// TwinCAT 3 PLC project Publisher
// ProgramVersion: 3.1.4022.0
// libraries:
//   Tc2_Standard, * (Beckhoff Automation GmbH)
//   Tc2_System, * (Beckhoff Automation GmbH)
//   Tc3_EventLogger, * (Beckhoff Automation GmbH)
//   Tc3_Module, * (Beckhoff Automation GmbH)
// project tree:
//   / PublisherTask.TcTTO (not stored)
//   POUs/ MAIN.TcPOU
// real-time tasks:
//   TASK PublisherTask: cycle T#10ms, priority 20, ADS port 350
//   TASK ListenerTask: cycle T#10ms, priority 1, ADS port 351

// ---- POUs/MAIN.TcPOU
PROGRAM MAIN
VAR
	bSendMessage : BOOL;
	bSendMessage_NotSubscribed: BOOL;
	bRaiseAlarm : BOOL;
	bConfirmAlarm : BOOL;
	bClearAlarm: BOOL;

	fbLogger : FB_TcEventLogger;
	fbMessage : FB_TcMessage;
	fbMessageArgs : FB_TcMessage;
	fbAlarm : FB_TcAlarm;
	bIsInitalized : BOOL;
	
	bSetJsonAttribute : BOOL;
	sJsonAttribute : STRING := '{"key":"value"}';
	
	hr : HRESULT;
	hrLastError : HRESULT;
	
	
	fbSource : FB_TcSourceInfo;
	bSendMessage_Win32ErrorClass: BOOL;
	bClearLoggedEvents: BOOL;
	bSendMessageWithArgs: BOOL;
END_VAR

IF NOT bIsInitalized THEN
	bIsInitalized := TRUE;
	hr := fbAlarm.CreateEx(TC_EVENTS.PublisherEventClass.Alarm, TRUE, 0);
	IF FAILED(hr) THEN
		hrLastError := hr;
	END_IF
	hr := fbMessage.CreateEx(TC_EVENTS.PublisherEventClass.Message, 0);
	IF FAILED(hr) THEN
		hrLastError := hr;
	END_IF
	hr := fbMessageArgs.CreateEx(TC_EVENTS.PublisherEventClass.MessageWithArgs, 0);
	IF FAILED(hr) THEN
		hrLastError := hr;
	END_IF
END_IF

IF bSetJsonAttribute THEN
	bSetJsonAttribute := FALSE;
	hr := fbAlarm.SetJsonAttribute(sJsonAttribute);
	IF FAILED(hr) THEN
		hrLastError := hr;
	END_IF
	hr := fbMessage.SetJsonAttribute(sJsonAttribute);
	IF FAILED(hr) THEN
		hrLastError := hr;
	END_IF
END_IF

IF bSendMessage THEN
	bSendMessage := FALSE;
	hr := fbMessage.Send(0);
	IF FAILED(hr) THEN
		hrLastError := hr;
	END_IF
END_IF

IF bSendMessageWithArgs THEN
	bSendMessageWithArgs := FALSE;
	//Using a String means to use a fixed String which cant be translated by a HMI. 
	//If you want to have translated arguments you could make use of referenced events like shown here. They have their own translations available. 
	fbMessageArgs.ipArguments.Clear().AddDInt(42).AddString('abc').AddEventReferenceEx(TC_EVENTS.PublisherEventClass.ReferencedEvent).AddString('AppendedArgument'); 
	hr := fbMessageArgs.Send(0);
	IF FAILED(hr) THEN
		hrLastError := hr;
	END_IF
END_IF

IF bSendMessage_NotSubscribed THEN
	bSendMessage_NotSubscribed := FALSE;
	fbSource.sName := 'Not subscribed Event';
	hr := fbLogger.SendMessageEx(TC_EVENTS.AnotherEventClass.NonSubscribedEvent, 0,0,0);
	IF FAILED(hr) THEN
		hrLastError := hr;
	END_IF
END_IF

IF bSendMessage_Win32ErrorClass THEN //use a TwinCAT provided Eventclass
	bSendMessage_Win32ErrorClass := FALSE;
	fbSource.sName := 'TwinCAT provided event';
	hr := fbLogger.SendMessageEx(TC_EVENTS.Win32EventClass.ERROR_SUCCESS, 0,0,0);
	IF FAILED(hr) THEN
		hrLastError := hr;
	END_IF
END_IF

IF bRaiseAlarm THEN
	bRaiseAlarm := FALSE;
	hr := fbAlarm.Raise(0);
	IF FAILED(hr) THEN
		hrLastError := hr;
	END_IF
END_IF

IF bConfirmAlarm THEN
	bConfirmAlarm := FALSE;
	hr := fbAlarm.Confirm(0);
	IF FAILED(hr) THEN
		hrLastError := hr;
	END_IF
END_IF

IF bClearAlarm THEN
	bClearAlarm := FALSE;
	hr := fbAlarm.Clear(0, FALSE);
	IF FAILED(hr) THEN
		hrLastError := hr;
	END_IF
END_IF

END_PROGRAM
